Staubli VAL3: InitRobot.pgx

program InitRobot()
  local num maxSpeed
  local num cpt
begin
//*******************************************************************************
//*   ______
//*  / _____) /|
//* | |      / /
//* | | /\  / /
//* | | \ \/ /  _      Copyright (c) KEOLABS, 2016
//* | |  \__/  | |        http://www.keolabs.com
//* | |________| |
//*  \__________/
//*
//********************************************************************************
//*@file          : InitRobot
//*@author        : Yves Ragot
//*@version       : $Id: InitRobot.pgx 1658 2017-01-25 07:36:52Z yves $
//*@brief         : InitRobot command treatment
//*
//*******************************************************************************/

  // reinit default values
  call Init()

  // remote ?
  if (workingMode() != 4)
      popUpMsg("Please switch to remote mode")
      GeneralStatus = 106
  else
      // auto connection mouvement in remote mode
      autoConnectMove(true)

      // reset motion task
      resetMotion()

      // power
      enablePower()
      cpt = 0
      do
        delay(0.1)
        cpt = cpt + 1
      until (isPowered() or (cpt >  50))

      if (cpt > 50)
          GeneralStatus = 106
      else
          //set max speed
          maxSpeed = getMonitorSpeed()
          if (maxSpeed < 100)
              setMonitorSpeed(100)
          endIf
      endIf
  endIf
end
